(*			
	EVERDE sp. z o.o.
	Rafał Osajda		31.01.2025		TC 4026.13		wer. 0.0.0.1
	Obsługa przycisku ze stykiem NC
*)
FUNCTION_BLOCK FB_IOButton_NC EXTENDS FB_IOButton
VAR
END_VAR

METHOD FB_init : BOOL
VAR_INPUT
	bInitRetains : BOOL; // if TRUE, the retain variables are initialized (warm start / cold start)
	bInCopyCode : BOOL;  // if TRUE, the instance afterwards gets moved into the copy code (online change)
END_VAR
THIS^.bContactPrev		:= TRUE;
END_METHOD

METHOD PUBLIC GetRisingEdgePressed : BOOL
VAR_INPUT
END_VAR
IF (THIS^.bContactPrev AND NOT THIS^.bContact) THEN
	THIS^.bContactPrev		:= FALSE;
	GetRisingEdgePressed	:= TRUE;
ELSIF (NOT THIS^.bContactPrev AND THIS^.bContact) THEN
	THIS^.bContactPrev		:= TRUE;
END_IF
END_METHOD

(*			
	EVERDE sp. z o.o.
	Rafał Osajda		31.01.2025		TC 4026.13		wer. 0.0.0.1
	Zwraca stan przycisku
*)
METHOD IsPressed : BOOL
IsPressed			:= NOT THIS^.bContact;
END_METHOD

END_FUNCTION_BLOCK

(* stored: Version 1.1.0.1
   POU FB_IOButton_NC: Id {67ab5e68-7c00-41fd-bce3-35b5b14f6170}, SpecialFunc None
   Method FB_init: Id {bc349bf6-7b48-0928-3da6-6428e4f7ef16}
   Method GetRisingEdgePressed: Id {b870440c-9fe7-0516-34cf-751334598583}
   Method IsPressed: Id {10c67b5f-8f1a-4820-9165-12fe0c243f33} *)
